# EPICS substitutions: apps/caenHv527App/Db/dchvWaveforms-S126.substitutions
file "db/dchvWaveforms.db" {
  pattern { S, R, L }
  { 1, 1, 1 }
  { 1, 1, 2 }
  { 1, 2, 3 }
  { 1, 2, 4 }
  { 1, 3, 5 }
  { 1, 3, 6 }
  { 2, 1, 1 }
  { 2, 1, 2 }
  { 2, 2, 3 }
  { 2, 2, 4 }
  { 2, 3, 5 }
  { 2, 3, 6 }
  { 6, 1, 1 }
  { 6, 1, 2 }
  { 6, 2, 3 }
  { 6, 2, 4 }
  { 6, 3, 5 }
  { 6, 3, 6 }
}
